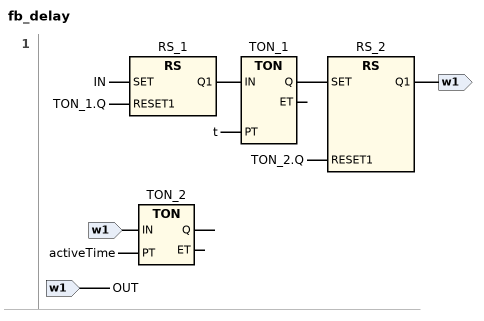
// NETWORK 1
RS_1(SET := IN, RESET1 := TON_1.Q); // RS
TON_1(IN := RS_1.Q1, PT := t); // TON
RS_2(SET := TON_1.Q, RESET1 := TON_2.Q); // RS
TON_2(IN := RS_2.Q1, PT := activeTime); // TON
OUT := RS_2.Q1;

END_FUNCTION_BLOCK

// Device/Application/functions/FB_CLK
// 50 % CLK heigh
FUNCTION_BLOCK FB_CLK
VAR_INPUT
	enable : BOOL := TRUE;
	CLK_Time : TIME := T#1s;
END_VAR
VAR
	RS_0: RS;
	TON_0: TON;
	RS_1: RS;
	TON_1: TON;
END_VAR
VAR_OUTPUT
	CLK :BOOL;
END_VAR

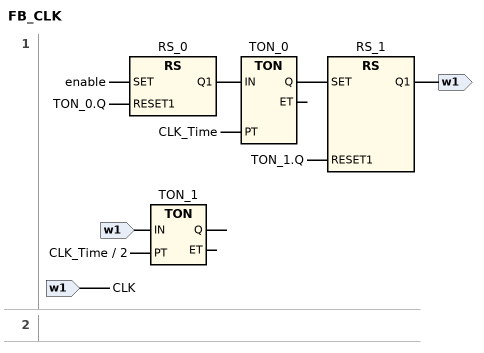
// NETWORK 1
RS_0(SET := enable, RESET1 := TON_0.Q); // RS
TON_0(IN := RS_0.Q1, PT := CLK_Time); // TON
RS_1(SET := TON_0.Q, RESET1 := TON_1.Q); // RS
TON_1(IN := RS_1.Q1, PT := CLK_Time / 2); // TON
CLK := RS_1.Q1;

// NETWORK 2

END_FUNCTION_BLOCK

// Device/Application/functions/Advanced_CTUD
FUNCTION_BLOCK Advanced_CTUD
VAR_INPUT
	CU: BOOL; //key
	CD: BOOL; //key
	activate: BOOL; // exmaple: index = 3 then true.
	frame: USINT; // frame where the button is
	reset : BOOL := 0; // reset to countValue before submit
	//submit : BOOL:= TRUE; // currently not working key or anything else, you can use trigger to make countedValue = newValue
	minValue : INT;
	maxValue: INT;
	countedValue: UINT;
END_VAR
VAR_OUTPUT
	newValue: UINT;
	active : BOOL;
END_VAR
VAR
	FB_smoothCLK_CU: FB_smoothCLK;
	FB_smoothCLK_CD: FB_smoothCLK;
	CTUD_Value: CTUD;
	SR_Changed: SR;
	MIN_1: BOOL;
END_VAR

VAR_IN_OUT

END_VAR
VAR // added by the converter: edge detectors and wires of the graphical bodies
    _rt1, _rt2, _rt3, _rt4, _rt5, _rt6, _rt7 : R_TRIG;
END_VAR

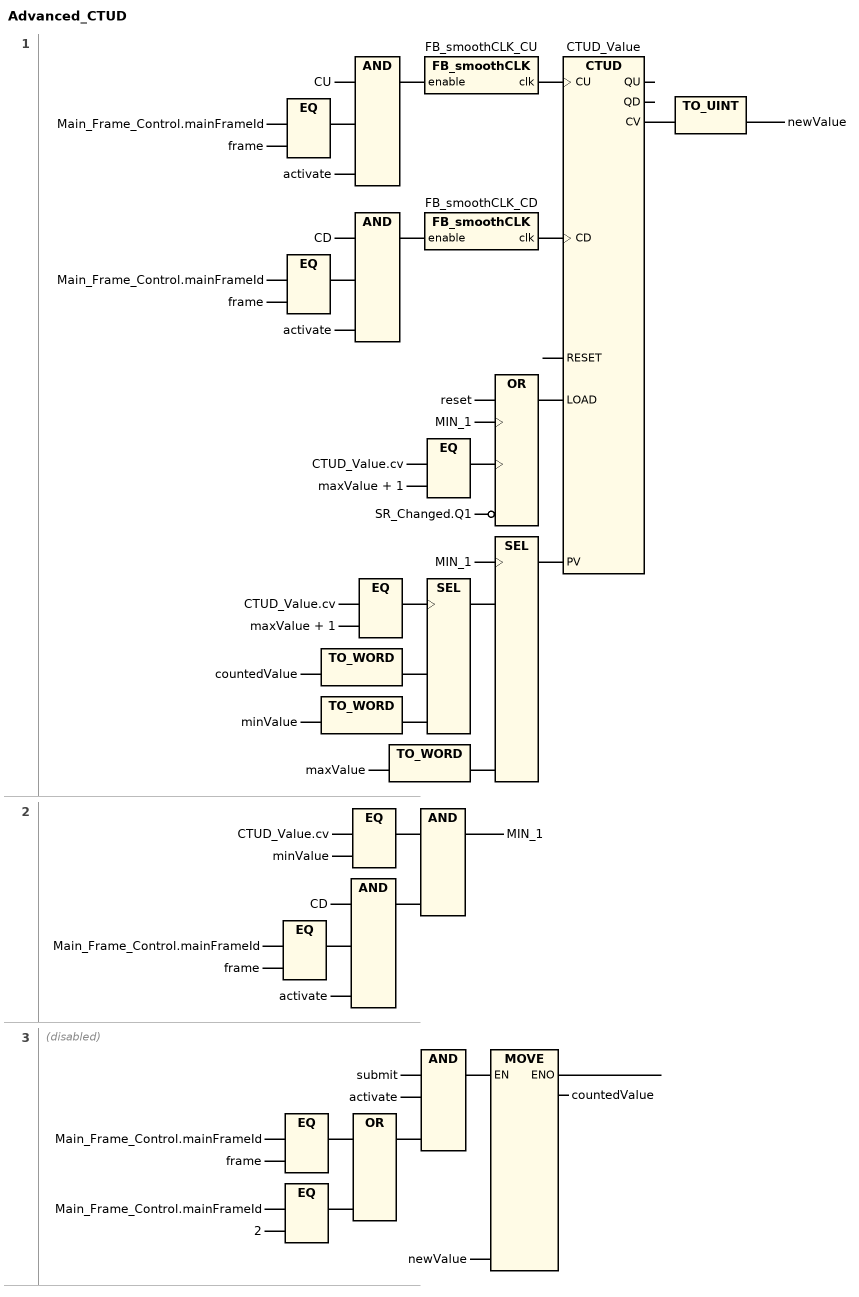
// NETWORK 1
FB_smoothCLK_CU(enable := CU AND Main_Frame_Control.mainFrameId = frame AND activate); // FB_smoothCLK
_rt1(CLK := FB_smoothCLK_CU.clk);
FB_smoothCLK_CD(enable := CD AND Main_Frame_Control.mainFrameId = frame AND activate); // FB_smoothCLK
_rt2(CLK := FB_smoothCLK_CD.clk);
_rt3(CLK := MIN_1);
_rt4(CLK := CTUD_Value.cv = (maxValue + 1));
_rt5(CLK := MIN_1);
_rt6(CLK := CTUD_Value.cv = (maxValue + 1));
CTUD_Value(
    CU := _rt1.Q,
    CD := _rt2.Q,
    LOAD := reset OR _rt3.Q OR _rt4.Q OR NOT SR_Changed.Q1,
    PV := SEL(_rt5.Q, SEL(_rt6.Q, TO_WORD(countedValue), TO_WORD(minValue)), TO_WORD(maxValue))); // CTUD
newValue := TO_UINT(CTUD_Value.CV);

// NETWORK 2
MIN_1 := CTUD_Value.cv = minValue AND (CD AND Main_Frame_Control.mainFrameId = frame AND activate);

// NETWORK 3 (disabled)
// IF submit AND activate AND (Main_Frame_Control.mainFrameId = frame OR Main_Frame_Control.mainFrameId = 2) THEN
//     countedValue := newValue;
// END_IF

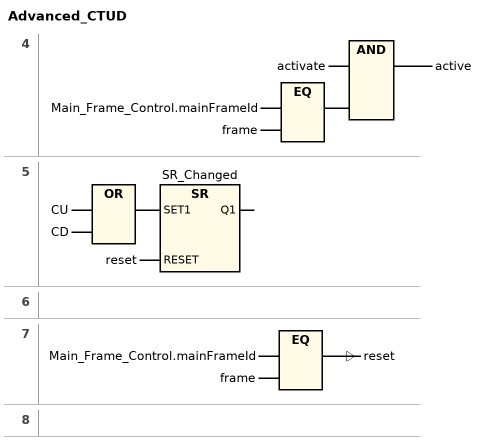
// NETWORK 4
active := activate AND Main_Frame_Control.mainFrameId = frame;

// NETWORK 5
SR_Changed(SET1 := CU OR CD, RESET := reset); // SR

// NETWORK 6

// NETWORK 7
_rt7(CLK := Main_Frame_Control.mainFrameId = frame);
reset := _rt7.Q;

// NETWORK 8

END_FUNCTION_BLOCK

// Device/Application/functions/FB_smoothCLK
FUNCTION_BLOCK FB_smoothCLK
VAR_INPUT
	enable : BOOL := TRUE; // use the same variable wich you used to In- or decrement the value
	CLK_TimeMin : TIME := T#50MS;
	//v : TIME := T#100MS; // sekund^-1
END_VAR
VAR_OUTPUT
	clk: BOOL;
END_VAR
VAR
	FB_CLK_0: FB_CLK;
	CLK_Time: TIME := T#1000MS;
	CLK_Time_End: TIME;
	FB_CLK_1: FB_CLK;
END_VAR
VAR // added by the converter: edge detectors and wires of the graphical bodies
    _w1 : INT;
    _ft1 : F_TRIG;
END_VAR

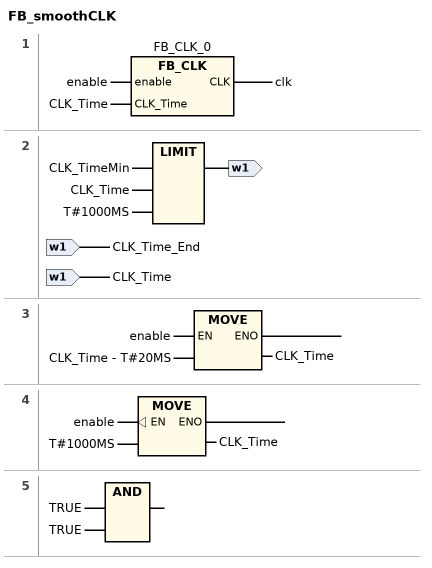
// NETWORK 1
FB_CLK_0(enable := enable, CLK_Time := CLK_Time); // FB_CLK
clk := FB_CLK_0.CLK;

// NETWORK 2
_w1 := LIMIT(CLK_TimeMin, CLK_Time, T#1000MS);
CLK_Time_End := _w1;
CLK_Time := _w1;

// NETWORK 3
IF enable THEN CLK_Time := CLK_Time - T#20MS; END_IF

// NETWORK 4
_ft1(CLK := enable);
IF _ft1.Q THEN CLK_Time := T#1000MS; END_IF

// NETWORK 5
(* TRUE AND TRUE; result not used *)

END_FUNCTION_BLOCK

// Device/Application/FBs/Paramater/parameterUpdate
FUNCTION_BLOCK parameterUpdate
VAR_INPUT
	EN: BOOL;
	selectedParameterIndex: INT;
END_VAR
VAR_OUTPUT


	iDistanceBetweenRowsInMeter: REAL:= 1.5;
	iDistanceBeforInMeter: REAL:= 1.5;
	iDistanceAfterInMeter: REAL:= 1.5;
	iCountRows: USINT:=15 ;
	strRowsDirection: STRING;
	bRowsDirection: BOOL;
	
END_VAR
VAR
	CTU_LeftRight: CTU;
	FB_ChangeDistance_CountRows: FB_UpdatingDistanceParameter;
	FB_ChangeDistance_AfterInMeter: FB_UpdatingDistanceParameter;
	FB_ChangeDistance_BeforInMeter: FB_UpdatingDistanceParameter;
	FB_ChangeDistance_BetweenInMeter: FB_UpdatingDistanceParameter;
	rCountRows: REAL;
	TOGGLE_0:TOGGLE;
	TON_CLK: TON;
	RS_CLK: RS;

	// Row Parameter

	CLK_PULSE_0: CLK_PULSE;
	RS_CLK2: RS;
	TON_CLK2: TON;
END_VAR

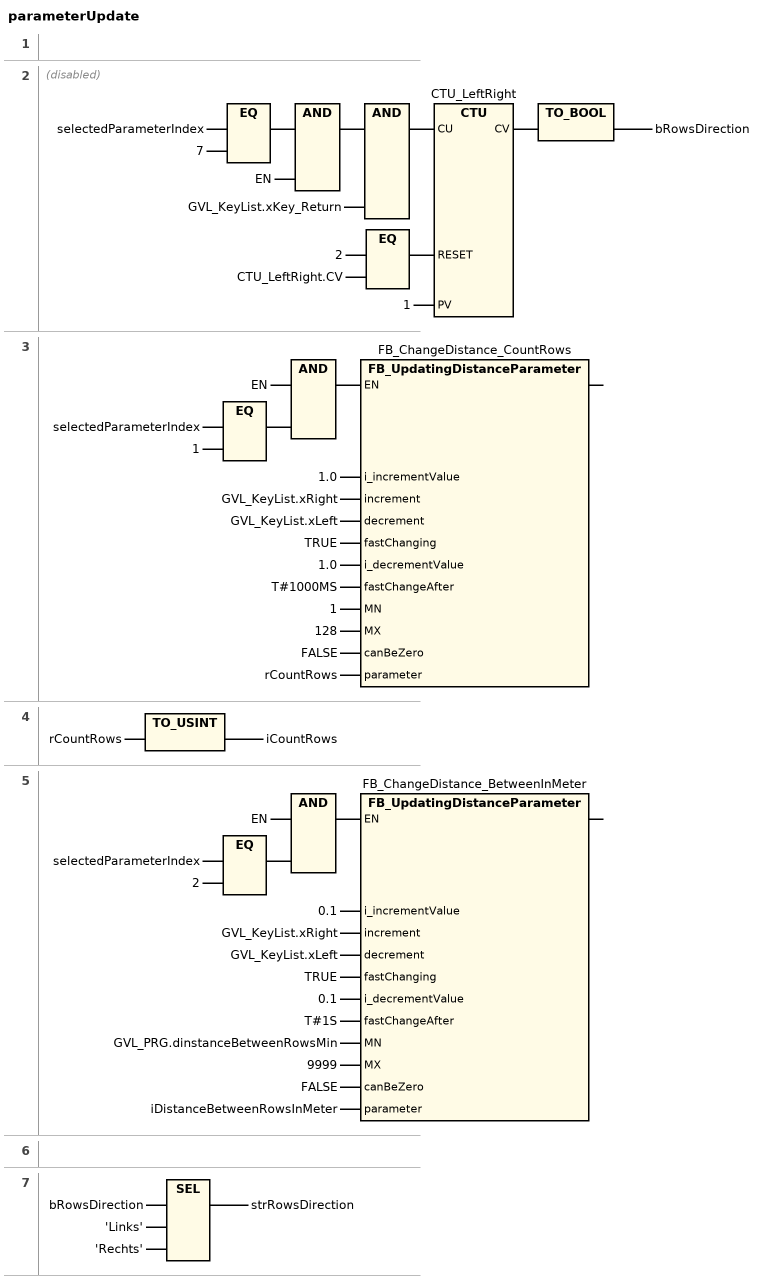
// NETWORK 1

// NETWORK 2 (disabled)
// CTU_LeftRight(
//     CU := (selectedParameterIndex = 7 AND EN) AND GVL_KeyList.xKey_Return,
//     RESET := 2 = CTU_LeftRight.CV,
//     PV := 1); // CTU
// bRowsDirection := TO_BOOL(CTU_LeftRight.CV);

// NETWORK 3
FB_ChangeDistance_CountRows(
    EN := EN AND selectedParameterIndex = 1,
    i_incrementValue := 1.0,
    increment := GVL_KeyList.xRight,
    decrement := GVL_KeyList.xLeft,
    fastChanging := TRUE,
    i_decrementValue := 1.0,
    fastChangeAfter := T#1000MS,
    MN := 1,
    MX := 128,
    canBeZero := FALSE,
    parameter := rCountRows); // FB_UpdatingDistanceParameter

// NETWORK 4
iCountRows := TO_USINT(rCountRows);

// NETWORK 5
FB_ChangeDistance_BetweenInMeter(
    EN := EN AND selectedParameterIndex = 2,
    i_incrementValue := 0.1,
    increment := GVL_KeyList.xRight,
    decrement := GVL_KeyList.xLeft,
    fastChanging := TRUE,
    i_decrementValue := 0.1,
    fastChangeAfter := T#1S,
    MN := GVL_PRG.dinstanceBetweenRowsMin,
    MX := 9999,
    canBeZero := FALSE,
    parameter := iDistanceBetweenRowsInMeter); // FB_UpdatingDistanceParameter

// NETWORK 6

// NETWORK 7
strRowsDirection := SEL(bRowsDirection, 'Links', 'Rechts');

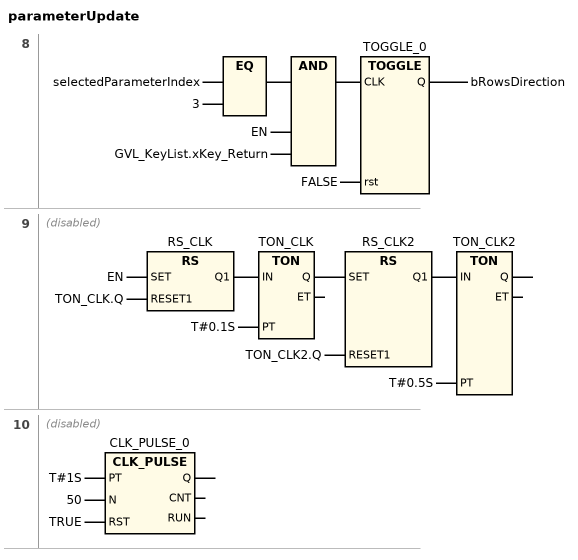
// NETWORK 8
TOGGLE_0(CLK := selectedParameterIndex = 3 AND EN AND GVL_KeyList.xKey_Return, rst := FALSE); // TOGGLE
bRowsDirection := TOGGLE_0.Q;

// NETWORK 9 (disabled)
// RS_CLK(SET := EN, RESET1 := TON_CLK.Q); // RS
// TON_CLK(IN := RS_CLK.Q1, PT := T#0.1S); // TON
// RS_CLK2(SET := TON_CLK.Q, RESET1 := TON_CLK2.Q); // RS
// TON_CLK2(IN := RS_CLK2.Q1, PT := T#0.5S); // TON

// NETWORK 10 (disabled)
// CLK_PULSE_0(PT := T#1S, N := 50, RST := TRUE); // CLK_PULSE

END_FUNCTION_BLOCK

// Device/Application/FBs/Paramater/FB_UpdatingDistanceParameter
FUNCTION_BLOCK FB_UpdatingDistanceParameter
VAR_INPUT
	EN: BOOL;
	i_incrementValue: REAL := 0.1;
	increment: BOOL := FALSE;
	decrement: BOOL := FALSE;
	fastChanging: BOOL := TRUE;
	i_decrementValue: REAL := 0.1;
	fastChangeAfter: TIME:= T#1S;
	MN: REAL := 0;
	MX: REAL:= 9999;
	canBeZero: BOOL:= TRUE;
	
END_VAR
VAR_OUTPUT
END_VAR
VAR
	RS_CLK: RS;
	TON_CLK: TON;
	canBeZeroIfMnGreaterO: BOOL;
	TON_FastEditingDown: TON;
	TON_FastEditingUp: TON;
	canBeZeroIfMXLessThan0: BOOL;
	incrementValue: REAL;
	decrementValue: REAL;
END_VAR
VAR_IN_OUT
		parameter: REAL;
END_VAR
VAR // added by the converter: edge detectors and wires of the graphical bodies
    _w1, _w2, _w3, _w4 : BOOL;
    _rt1, _rt2, _rt3, _rt4 : R_TRIG;
END_VAR

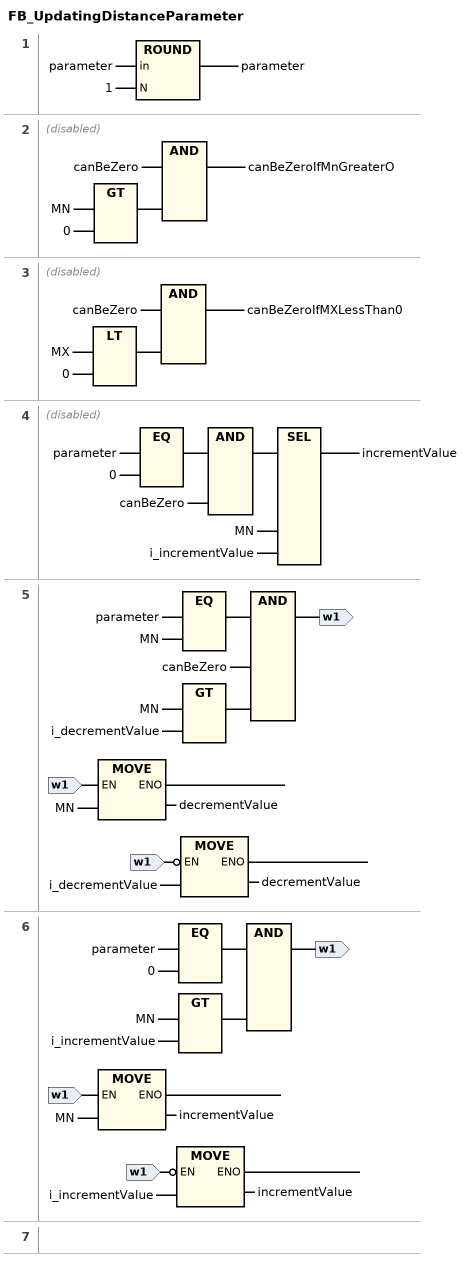
// NETWORK 1
parameter := ROUND(in := parameter, N := 1);

// NETWORK 2 (disabled)
// canBeZeroIfMnGreaterO := canBeZero AND MN > 0;

// NETWORK 3 (disabled)
// canBeZeroIfMXLessThan0 := canBeZero AND MX < 0;

// NETWORK 4 (disabled)
// incrementValue := SEL(parameter = 0 AND canBeZero, MN, i_incrementValue);

// NETWORK 5
_w1 := parameter = MN AND canBeZero AND MN > i_decrementValue;
IF _w1 THEN decrementValue := MN; END_IF
IF NOT _w1 THEN decrementValue := i_decrementValue; END_IF

// NETWORK 6
_w2 := parameter = 0 AND MN > i_incrementValue;
IF _w2 THEN incrementValue := MN; END_IF
IF NOT _w2 THEN incrementValue := i_incrementValue; END_IF

// NETWORK 7

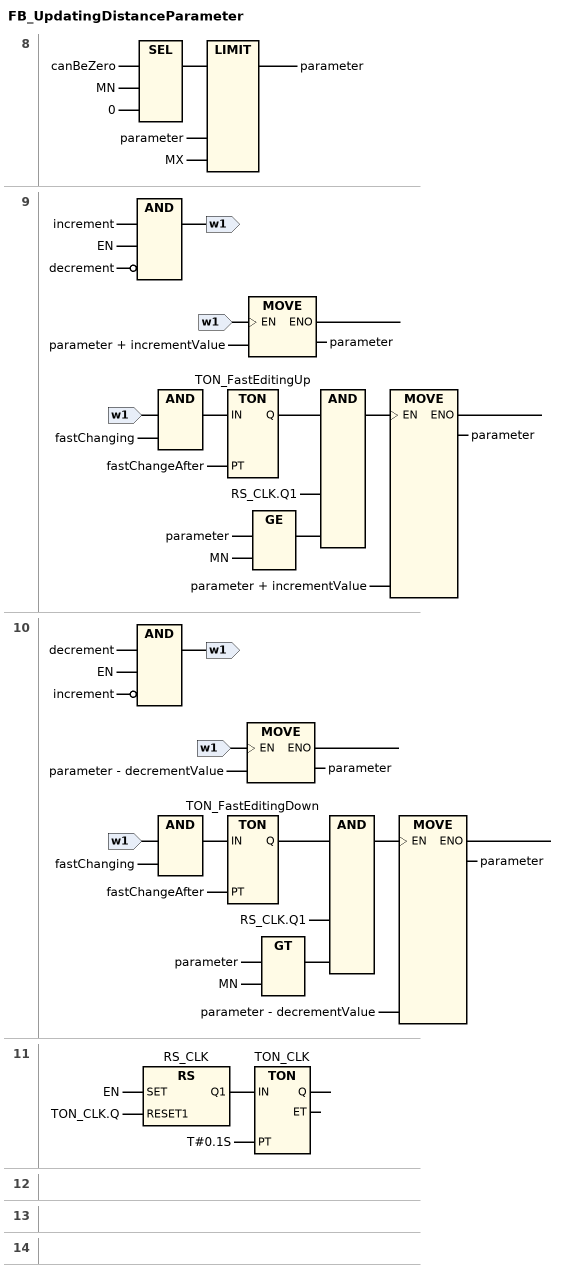
// NETWORK 8
parameter := LIMIT(SEL(canBeZero, MN, 0), parameter, MX);

// NETWORK 9
_w3 := increment AND EN AND NOT decrement;
_rt1(CLK := _w3);
IF _rt1.Q THEN parameter := parameter + incrementValue; END_IF
TON_FastEditingUp(IN := _w3 AND fastChanging, PT := fastChangeAfter); // TON
_rt2(CLK := TON_FastEditingUp.Q AND RS_CLK.Q1 AND parameter >= MN);
IF _rt2.Q THEN parameter := parameter + incrementValue; END_IF

// NETWORK 10
_w4 := decrement AND EN AND NOT increment;
_rt3(CLK := _w4);
IF _rt3.Q THEN parameter := parameter - decrementValue; END_IF
TON_FastEditingDown(IN := _w4 AND fastChanging, PT := fastChangeAfter); // TON
_rt4(CLK := TON_FastEditingDown.Q AND RS_CLK.Q1 AND parameter > MN);
IF _rt4.Q THEN parameter := parameter - decrementValue; END_IF

// NETWORK 11
RS_CLK(SET := EN, RESET1 := TON_CLK.Q); // RS
TON_CLK(IN := RS_CLK.Q1, PT := T#0.1S); // TON

// NETWORK 12

// NETWORK 13

// NETWORK 14

END_FUNCTION_BLOCK

// Device/Application/FBs/Controll/RoboterControl
FUNCTION_BLOCK RoboterControl
VAR_INPUT
	
	iCountRows:USINT;
	iDistanceAfterInMeter: REAL;
	iDistanceBeforInMeter: REAL;
	iDistanceBetweenRowsInMeter: REAL;
	bRowsDirection: BOOL;
END_VAR
VAR_OUTPUT
END_VAR
VAR
	AutomaticModeControl_0: AutomaticModeControl;
	PrepareAutomaticModeParameterForCAN_0: PrepareParameterForCAN;
END_VAR
VAR // added by the converter: edge detectors and wires of the graphical bodies
    _rt1, _rt2 : R_TRIG;
END_VAR

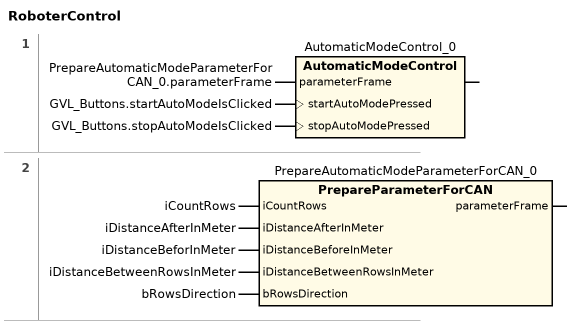
// NETWORK 1
_rt1(CLK := GVL_Buttons.startAutoModeIsClicked);
_rt2(CLK := GVL_Buttons.stopAutoModeIsClicked);
AutomaticModeControl_0(
    parameterFrame := PrepareAutomaticModeParameterForCAN_0.parameterFrame,
    startAutoModePressed := _rt1.Q,
    stopAutoModePressed := _rt2.Q); // AutomaticModeControl

// NETWORK 2
PrepareAutomaticModeParameterForCAN_0(
    iCountRows := iCountRows,
    iDistanceAfterInMeter := iDistanceAfterInMeter,
    iDistanceBeforeInMeter := iDistanceBeforInMeter,
    iDistanceBetweenRowsInMeter := iDistanceBetweenRowsInMeter,
    bRowsDirection := bRowsDirection); // PrepareParameterForCAN

END_FUNCTION_BLOCK

// Device/Application/FBs/Controll/AutomaticModeControl
FUNCTION_BLOCK AutomaticModeControl
VAR_INPUT
	parameterFrame: ARRAY[0..7] OF USINT;
	startAutoModePressed: BOOL;
	stopAutoModePressed: BOOL;
END_VAR
VAR_OUTPUT
END_VAR
VAR
	CAN_Tx_StartAutomode: ifmRCAN.CAN_Tx;
	CAN_Tx_StopAutoMode: ifmRCAN.CAN_Tx;
	CAN_Tx_PauseAutoMode: ifmRCAN.CAN_Tx;
	CAN_Tx_ResumeAutoMode: ifmRCAN.CAN_Tx;
	//AM_Paused: BOOL;
	CAN_Tx_ACK_Stop: ifmRCAN.CAN_Tx;
	SR_0: SR;
	SR_1: SR;
	rs_33: rs;
	CAN_Rx_jetson : ifmRCAN.CAN_Rx;
	SR_start_TX_State_Done: sr;
	fb_delay_1: FB_DELAY;
	FB_CLK_0: FB_CLK;
	test: BOOL;
	test1: BOOL;
	test2: BOOL;
	test4: BOOL;
	SR_waitingStartTime: sr;
	startNow: BOOL;
	test6: BOOL;
END_VAR
VAR // added by the converter: edge detectors and wires of the graphical bodies
    _rt1, _rt2, _rt3, _rt4, _rt5, _rt6, _rt7, _rt8, _rt9, _rt10, _rt11, _rt12, _rt13, _rt14 : R_TRIG;
    _ft1, _ft2, _ft3, _ft4, _ft5, _ft6, _ft7 : F_TRIG;
    _w1, _w2, _w3 : BOOL;
END_VAR

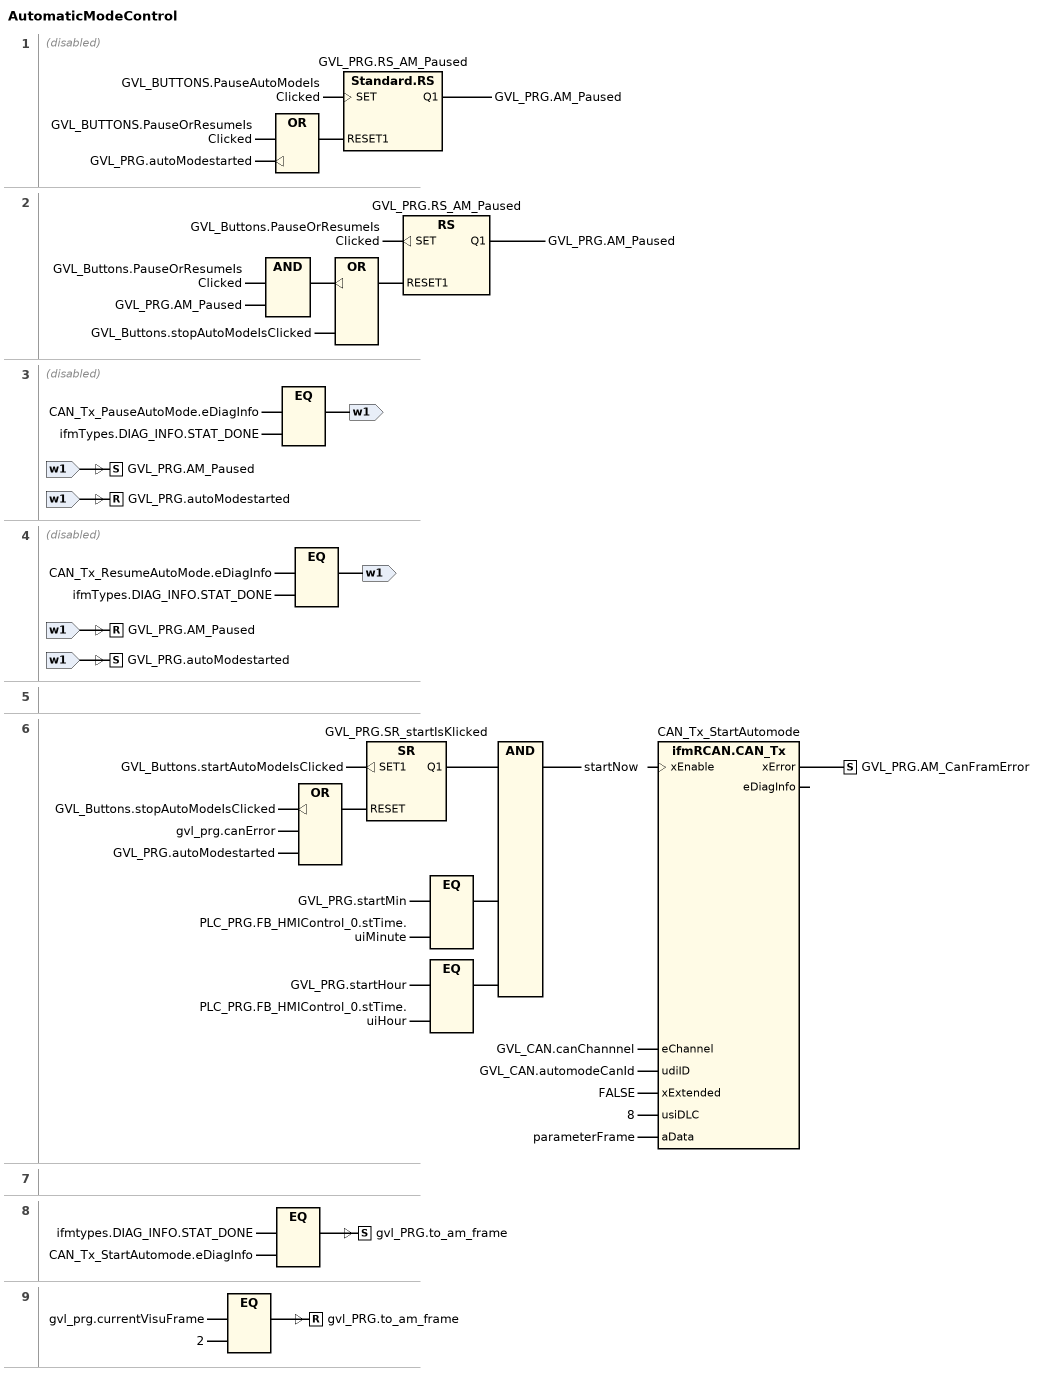
// NETWORK 1 (disabled)
// _rt1(CLK := GVL_BUTTONS.PauseAutoModeIsClicked);
// _ft1(CLK := GVL_PRG.autoModestarted);
// GVL_PRG.RS_AM_Paused(SET := _rt1.Q, RESET1 := GVL_BUTTONS.PauseOrResumeIsClicked OR _ft1.Q); // Standard.RS
// GVL_PRG.AM_Paused := GVL_PRG.RS_AM_Paused.Q1;

// NETWORK 2
_ft2(CLK := GVL_Buttons.PauseOrResumeIsClicked);
_ft3(CLK := GVL_Buttons.PauseOrResumeIsClicked AND GVL_PRG.AM_Paused);
GVL_PRG.RS_AM_Paused(SET := _ft2.Q, RESET1 := _ft3.Q OR GVL_Buttons.stopAutoModeIsClicked); // RS
GVL_PRG.AM_Paused := GVL_PRG.RS_AM_Paused.Q1;

// NETWORK 3 (disabled)
// _w1 := CAN_Tx_PauseAutoMode.eDiagInfo = ifmTypes.DIAG_INFO.STAT_DONE;
// _rt2(CLK := _w1);
// GVL_PRG.AM_Paused S= _rt2.Q;
// _rt3(CLK := _w1);
// GVL_PRG.autoModestarted R= _rt3.Q;

// NETWORK 4 (disabled)
// _w2 := CAN_Tx_ResumeAutoMode.eDiagInfo = ifmTypes.DIAG_INFO.STAT_DONE;
// _rt4(CLK := _w2);
// GVL_PRG.AM_Paused R= _rt4.Q;
// _rt5(CLK := _w2);
// GVL_PRG.autoModestarted S= _rt5.Q;

// NETWORK 5

// NETWORK 6
_ft4(CLK := GVL_Buttons.startAutoModeIsClicked);
_ft5(CLK := GVL_Buttons.stopAutoModeIsClicked);
GVL_PRG.SR_startIsKlicked(SET1 := _ft4.Q, RESET := _ft5.Q OR gvl_prg.canError OR GVL_PRG.autoModestarted); // SR
_w3 := GVL_PRG.SR_startIsKlicked.Q1 AND GVL_PRG.startMin = PLC_PRG.FB_HMIControl_0.stTime.uiMinute AND GVL_PRG.startHour = PLC_PRG.FB_HMIControl_0.stTime.uiHour;
startNow := _w3;
_rt6(CLK := _w3);
CAN_Tx_StartAutomode(
    xEnable := _rt6.Q,
    eChannel := GVL_CAN.canChannnel,
    udiID := GVL_CAN.automodeCanId,
    xExtended := FALSE,
    usiDLC := 8,
    aData := parameterFrame); // ifmRCAN.CAN_Tx
GVL_PRG.AM_CanFramError S= CAN_Tx_StartAutomode.xError;

// NETWORK 7

// NETWORK 8
_rt7(CLK := ifmtypes.DIAG_INFO.STAT_DONE = CAN_Tx_StartAutomode.eDiagInfo);
gvl_PRG.to_am_frame S= _rt7.Q;

// NETWORK 9
_rt8(CLK := gvl_prg.currentVisuFrame = 2);
gvl_PRG.to_am_frame R= _rt8.Q;

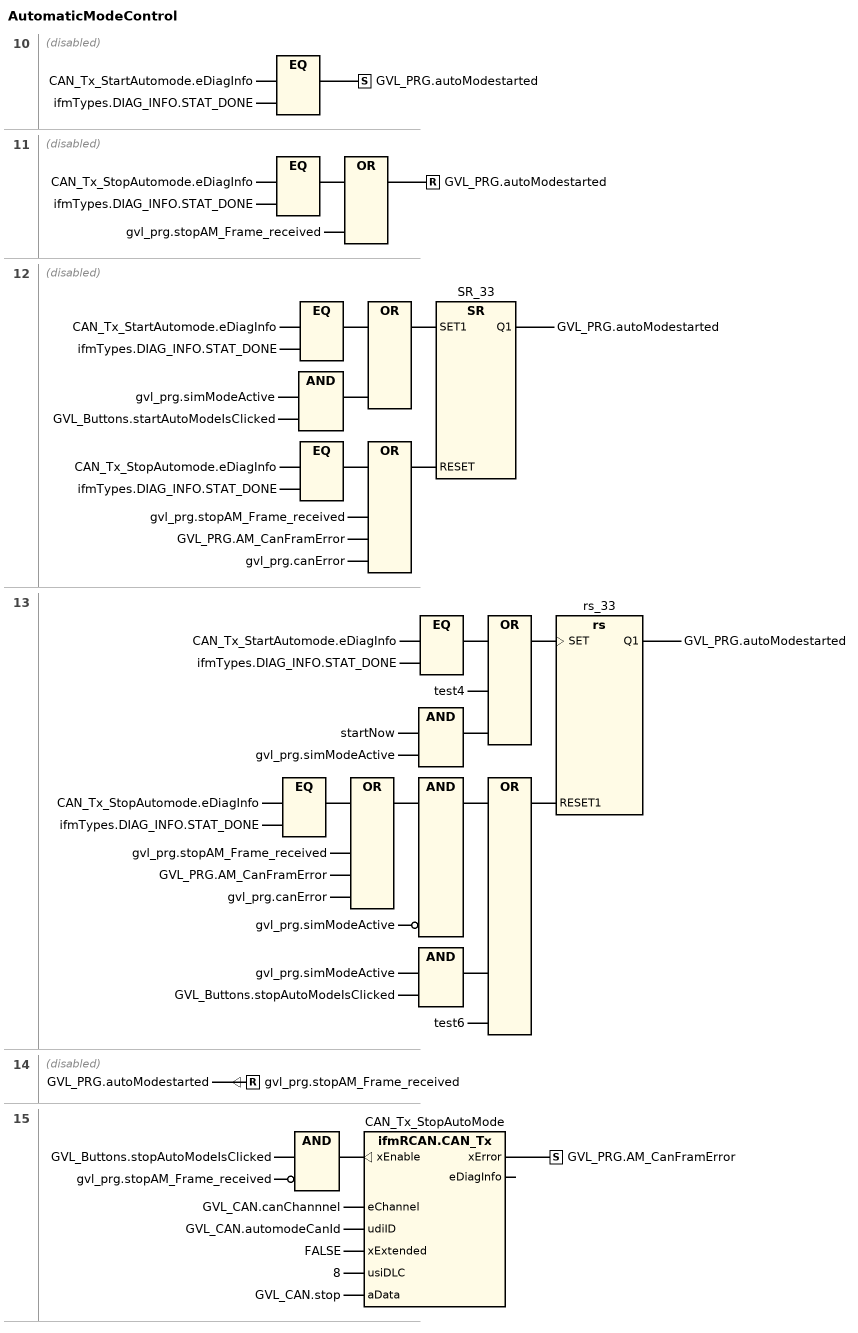
// NETWORK 10 (disabled)
// GVL_PRG.autoModestarted S= CAN_Tx_StartAutomode.eDiagInfo = ifmTypes.DIAG_INFO.STAT_DONE;

// NETWORK 11 (disabled)
// GVL_PRG.autoModestarted R= CAN_Tx_StopAutomode.eDiagInfo = ifmTypes.DIAG_INFO.STAT_DONE OR gvl_prg.stopAM_Frame_received;

// NETWORK 12 (disabled)
// SR_33(SET1 := CAN_Tx_StartAutomode.eDiagInfo = ifmTypes.DIAG_INFO.STAT_DONE OR gvl_prg.simModeActive AND GVL_Buttons.startAutoModeIsClicked, RESET := CAN_Tx_StopAutomode.eDiagInfo = ifmTypes.DIAG_INFO.STAT_DONE OR gvl_prg.stopAM_Frame_received OR GVL_PRG.AM_CanFramError OR gvl_prg.canError); // SR
// GVL_PRG.autoModestarted := SR_33.Q1;

// NETWORK 13
_rt9(CLK := CAN_Tx_StartAutomode.eDiagInfo = ifmTypes.DIAG_INFO.STAT_DONE OR test4 OR startNow AND gvl_prg.simModeActive);
rs_33(SET := _rt9.Q, RESET1 := (CAN_Tx_StopAutomode.eDiagInfo = ifmTypes.DIAG_INFO.STAT_DONE OR gvl_prg.stopAM_Frame_received OR GVL_PRG.AM_CanFramError OR gvl_prg.canError) AND NOT gvl_prg.simModeActive OR gvl_prg.simModeActive AND GVL_Buttons.stopAutoModeIsClicked OR test6); // rs
GVL_PRG.autoModestarted := rs_33.Q1;

// NETWORK 14 (disabled)
// _ft6(CLK := GVL_PRG.autoModestarted);
// gvl_prg.stopAM_Frame_received R= _ft6.Q;

// NETWORK 15
_ft7(CLK := GVL_Buttons.stopAutoModeIsClicked AND NOT gvl_prg.stopAM_Frame_received);
CAN_Tx_StopAutoMode(
    xEnable := _ft7.Q,
    eChannel := GVL_CAN.canChannnel,
    udiID := GVL_CAN.automodeCanId,
    xExtended := FALSE,
    usiDLC := 8,
    aData := GVL_CAN.stop); // ifmRCAN.CAN_Tx
GVL_PRG.AM_CanFramError S= CAN_Tx_StopAutoMode.xError;

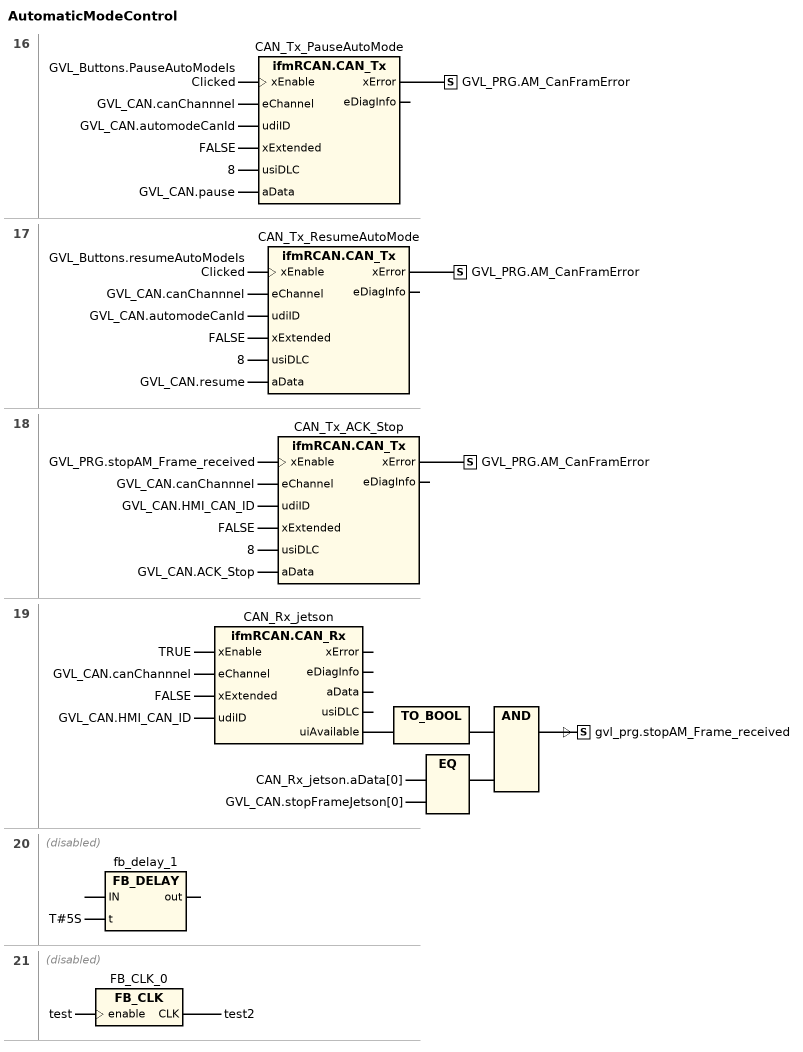
// NETWORK 16
_rt10(CLK := GVL_Buttons.PauseAutoModeIsClicked);
CAN_Tx_PauseAutoMode(
    xEnable := _rt10.Q,
    eChannel := GVL_CAN.canChannnel,
    udiID := GVL_CAN.automodeCanId,
    xExtended := FALSE,
    usiDLC := 8,
    aData := GVL_CAN.pause); // ifmRCAN.CAN_Tx
GVL_PRG.AM_CanFramError S= CAN_Tx_PauseAutoMode.xError;

// NETWORK 17
_rt11(CLK := GVL_Buttons.resumeAutoModeIsClicked);
CAN_Tx_ResumeAutoMode(
    xEnable := _rt11.Q,
    eChannel := GVL_CAN.canChannnel,
    udiID := GVL_CAN.automodeCanId,
    xExtended := FALSE,
    usiDLC := 8,
    aData := GVL_CAN.resume); // ifmRCAN.CAN_Tx
GVL_PRG.AM_CanFramError S= CAN_Tx_ResumeAutoMode.xError;

// NETWORK 18
_rt12(CLK := GVL_PRG.stopAM_Frame_received);
CAN_Tx_ACK_Stop(
    xEnable := _rt12.Q,
    eChannel := GVL_CAN.canChannnel,
    udiID := GVL_CAN.HMI_CAN_ID,
    xExtended := FALSE,
    usiDLC := 8,
    aData := GVL_CAN.ACK_Stop); // ifmRCAN.CAN_Tx
GVL_PRG.AM_CanFramError S= CAN_Tx_ACK_Stop.xError;

// NETWORK 19
CAN_Rx_jetson(
    xEnable := TRUE,
    eChannel := GVL_CAN.canChannnel,
    xExtended := FALSE,
    udiID := GVL_CAN.HMI_CAN_ID); // ifmRCAN.CAN_Rx
_rt13(CLK := TO_BOOL(CAN_Rx_jetson.uiAvailable) AND CAN_Rx_jetson.aData[0] = GVL_CAN.stopFrameJetson[0]);
gvl_prg.stopAM_Frame_received S= _rt13.Q;

// NETWORK 20 (disabled)
// fb_delay_1(t := T#5S); // FB_DELAY

// NETWORK 21 (disabled)
// _rt14(CLK := test);
// FB_CLK_0(enable := _rt14.Q); // FB_CLK
// test2 := FB_CLK_0.CLK;

END_FUNCTION_BLOCK

// Device/Application/FBs/Paramater/PrepareParameterForCAN
FUNCTION_BLOCK PrepareParameterForCAN
VAR_INPUT
	iCountRows:USINT;
	iDistanceAfterInMeter: REAL;
	iDistanceBeforeInMeter: REAL;
	iDistanceBetweenRowsInMeter: REAL;
	bRowsDirection: BOOL;
END_VAR
VAR_OUTPUT
	parameterFrame: ARRAY[0..7] OF USINT:=[0,0,0,0,0,0,0,0];
END_VAR
VAR
	iDistanceAfterInDM: USINT;
	iDistanceBeforeInDM: USINT;
	iDistanceBetweenRowsInDm: USINT;
	iRowsDirection: USINT;
	TO_ARRAY_Parameter: TO_ArrayOfUsint;
	TO_ArrayOfUsint_0: TO_ArrayOfUsint;
END_VAR

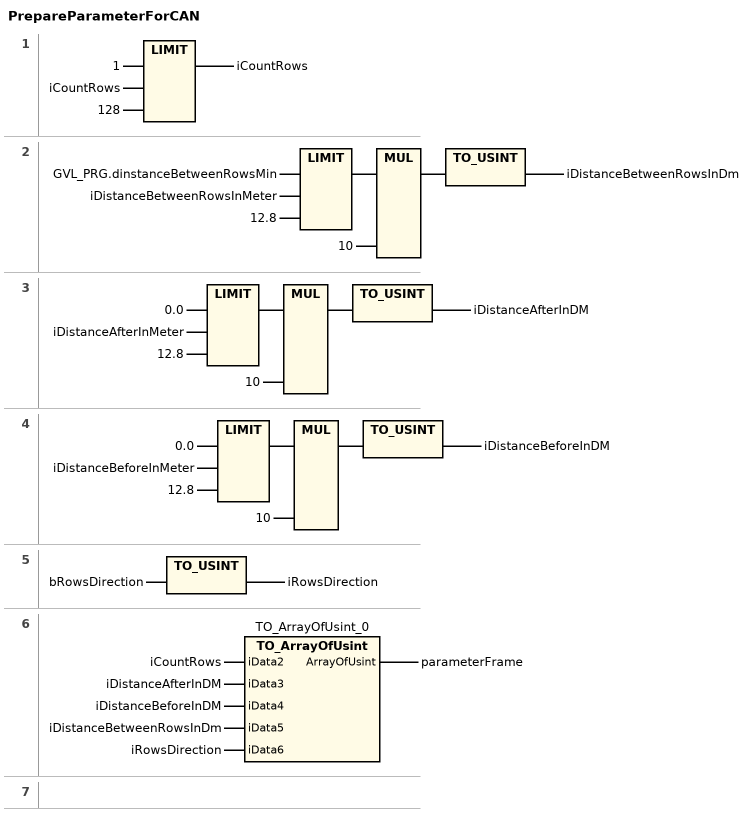
// NETWORK 1
iCountRows := LIMIT(1, iCountRows, 128);

// NETWORK 2
iDistanceBetweenRowsInDm := TO_USINT(LIMIT(GVL_PRG.dinstanceBetweenRowsMin, iDistanceBetweenRowsInMeter, 12.8) * 10);

// NETWORK 3
iDistanceAfterInDM := TO_USINT(LIMIT(0.0, iDistanceAfterInMeter, 12.8) * 10);

// NETWORK 4
iDistanceBeforeInDM := TO_USINT(LIMIT(0.0, iDistanceBeforeInMeter, 12.8) * 10);

// NETWORK 5
iRowsDirection := TO_USINT(bRowsDirection);

// NETWORK 6
TO_ArrayOfUsint_0(
    iData2 := iCountRows,
    iData3 := iDistanceAfterInDM,
    iData4 := iDistanceBeforeInDM,
    iData5 := iDistanceBetweenRowsInDm,
    iData6 := iRowsDirection); // TO_ArrayOfUsint
parameterFrame := TO_ArrayOfUsint_0.ArrayOfUsint;

// NETWORK 7

END_FUNCTION_BLOCK

// Device/Application/FBs/Paramater/TO_ArrayOfUsint
FUNCTION_BLOCK TO_ArrayOfUsint
VAR_INPUT
	iData1 : USINT := 0;
	iData2 : USINT := 0;
	iData3 : USINT := 0;
	iData4 : USINT := 0;
	iData5 : USINT := 0;
	iData6 : USINT := 0;
	iData7 : USINT := 0;
	iData8 : USINT := 0;
END_VAR
VAR_OUTPUT
	ArrayOfUsint: ARRAY [1..8] OF USINT;
END_VAR
VAR
END_VAR

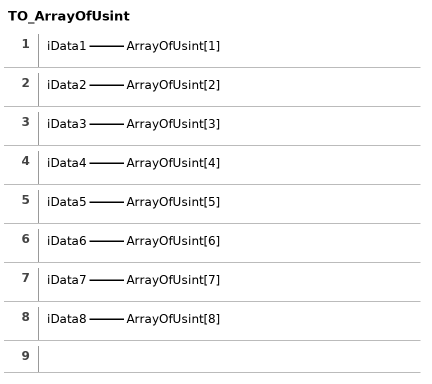
// NETWORK 1
ArrayOfUsint[1] := iData1;

// NETWORK 2
ArrayOfUsint[2] := iData2;

// NETWORK 3
ArrayOfUsint[3] := iData3;

// NETWORK 4
ArrayOfUsint[4] := iData4;

// NETWORK 5
ArrayOfUsint[5] := iData5;

// NETWORK 6
ArrayOfUsint[6] := iData6;

// NETWORK 7
ArrayOfUsint[7] := iData7;

// NETWORK 8
ArrayOfUsint[8] := iData8;

// NETWORK 9

END_FUNCTION_BLOCK

// Device/Application/FBs/Controll/SprayerControl
FUNCTION_BLOCK SprayerControl
VAR_INPUT
	//EN: BOOL;
		selectedParameterIndex: INT;
END_VAR
VAR_OUTPUT
END_VAR
VAR
	CAN_Tx_SprayerStartUp: ifmRCAN.CAN_Tx;
	CAN_Tx_SprayerStopUp: ifmRCAN.CAN_Tx;
	CAN_Tx_SprayerStartDown: ifmRCAN.CAN_Tx;
	CAN_Tx_SprayerStopDown: ifmRCAN.CAN_Tx;

	CAN_Tx_StopSprayer_1: ifmRCAN.CAN_Tx;
	CAN_Tx_StopSprayer_2: ifmRCAN.CAN_Tx;
	CAN_Tx_StopSprayer_3: ifmRCAN.CAN_Tx;
	
	CAN_Tx_PauseSprayer_1: ifmRCAN.CAN_Tx;
	CAN_Tx_PauseSprayer_2: ifmRCAN.CAN_Tx;
	CAN_Tx_PauseSprayer_3: ifmRCAN.CAN_Tx;
	
	CAN_Tx_ResumeSprayer_1: ifmRCAN.CAN_Tx;
	CAN_Tx_ResumeSprayer_2: ifmRCAN.CAN_Tx;
	CAN_Tx_ResumeSprayer_3: ifmRCAN.CAN_Tx;
	CAN_Tx_PumpOn: ifmRCAN.CAN_Tx;
	CAN_Tx_PumpOff: ifmRCAN.CAN_Tx;
	CAN_Tx_spryerLeftOn: ifmRCAN.CAN_Tx;
	CAN_Tx_spryerLeftOff: ifmRCAN.CAN_Tx;
	CAN_Tx_spryerRightOn: ifmRCAN.CAN_Tx;
	CAN_Tx_spryerRightOff: ifmRCAN.CAN_Tx;
END_VAR
VAR // added by the converter: edge detectors and wires of the graphical bodies
    _rt1, _rt2, _rt3, _rt4, _rt5, _rt6, _rt7, _rt8, _rt9, _rt10, _rt11, _rt12, _rt13 : R_TRIG;
    _ft1, _ft2, _ft3, _ft4, _ft5, _ft6 : F_TRIG;
END_VAR

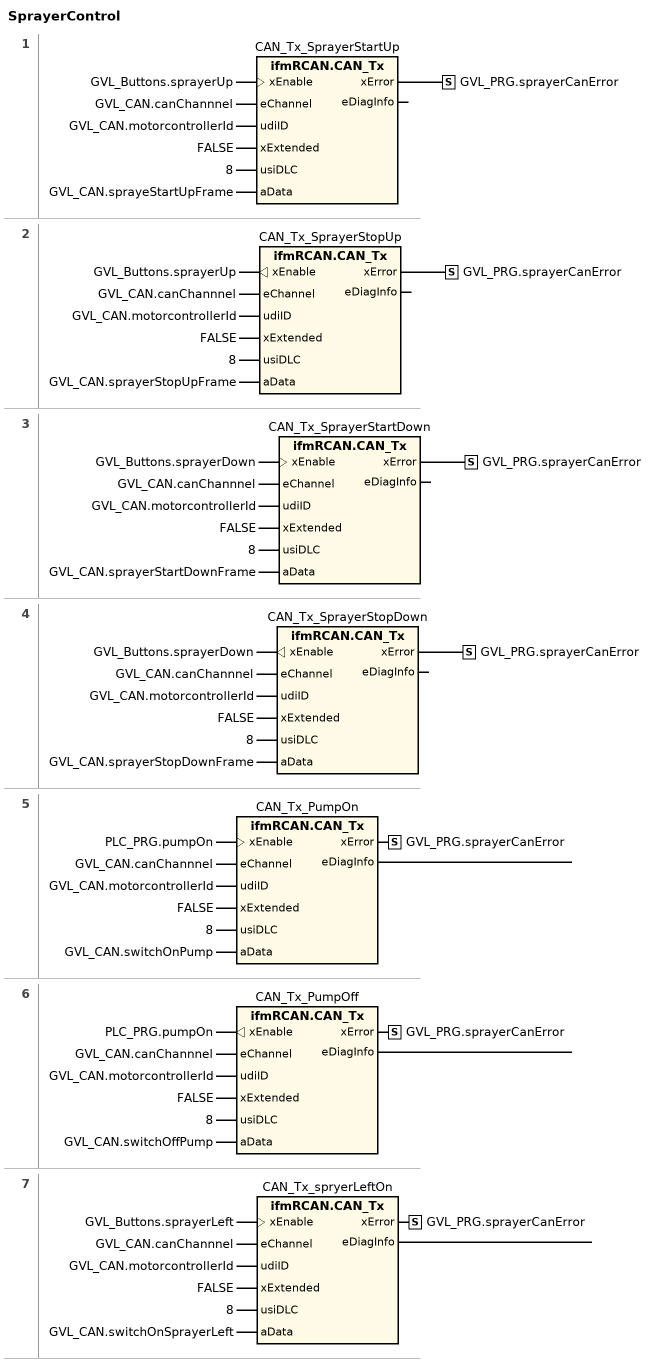
// NETWORK 1
_rt1(CLK := GVL_Buttons.sprayerUp);
CAN_Tx_SprayerStartUp(
    xEnable := _rt1.Q,
    eChannel := GVL_CAN.canChannnel,
    udiID := GVL_CAN.motorcontrollerId,
    xExtended := FALSE,
    usiDLC := 8,
    aData := GVL_CAN.sprayeStartUpFrame); // ifmRCAN.CAN_Tx
GVL_PRG.sprayerCanError S= CAN_Tx_SprayerStartUp.xError;

// NETWORK 2
_ft1(CLK := GVL_Buttons.sprayerUp);
CAN_Tx_SprayerStopUp(
    xEnable := _ft1.Q,
    eChannel := GVL_CAN.canChannnel,
    udiID := GVL_CAN.motorcontrollerId,
    xExtended := FALSE,
    usiDLC := 8,
    aData := GVL_CAN.sprayerStopUpFrame); // ifmRCAN.CAN_Tx
GVL_PRG.sprayerCanError S= CAN_Tx_SprayerStopUp.xError;

// NETWORK 3
_rt2(CLK := GVL_Buttons.sprayerDown);
CAN_Tx_SprayerStartDown(
    xEnable := _rt2.Q,
    eChannel := GVL_CAN.canChannnel,
    udiID := GVL_CAN.motorcontrollerId,
    xExtended := FALSE,
    usiDLC := 8,
    aData := GVL_CAN.sprayerStartDownFrame); // ifmRCAN.CAN_Tx
GVL_PRG.sprayerCanError S= CAN_Tx_SprayerStartDown.xError;

// NETWORK 4
_ft2(CLK := GVL_Buttons.sprayerDown);
CAN_Tx_SprayerStopDown(
    xEnable := _ft2.Q,
    eChannel := GVL_CAN.canChannnel,
    udiID := GVL_CAN.motorcontrollerId,
    xExtended := FALSE,
    usiDLC := 8,
    aData := GVL_CAN.sprayerStopDownFrame); // ifmRCAN.CAN_Tx
GVL_PRG.sprayerCanError S= CAN_Tx_SprayerStopDown.xError;

// NETWORK 5
_rt3(CLK := PLC_PRG.pumpOn);
CAN_Tx_PumpOn(
    xEnable := _rt3.Q,
    eChannel := GVL_CAN.canChannnel,
    udiID := GVL_CAN.motorcontrollerId,
    xExtended := FALSE,
    usiDLC := 8,
    aData := GVL_CAN.switchOnPump); // ifmRCAN.CAN_Tx
GVL_PRG.sprayerCanError S= CAN_Tx_PumpOn.xError;

// NETWORK 6
_ft3(CLK := PLC_PRG.pumpOn);
CAN_Tx_PumpOff(
    xEnable := _ft3.Q,
    eChannel := GVL_CAN.canChannnel,
    udiID := GVL_CAN.motorcontrollerId,
    xExtended := FALSE,
    usiDLC := 8,
    aData := GVL_CAN.switchOffPump); // ifmRCAN.CAN_Tx
GVL_PRG.sprayerCanError S= CAN_Tx_PumpOff.xError;

// NETWORK 7
_rt4(CLK := GVL_Buttons.sprayerLeft);
CAN_Tx_spryerLeftOn(
    xEnable := _rt4.Q,
    eChannel := GVL_CAN.canChannnel,
    udiID := GVL_CAN.motorcontrollerId,
    xExtended := FALSE,
    usiDLC := 8,
    aData := GVL_CAN.switchOnSprayerLeft); // ifmRCAN.CAN_Tx
GVL_PRG.sprayerCanError S= CAN_Tx_spryerLeftOn.xError;

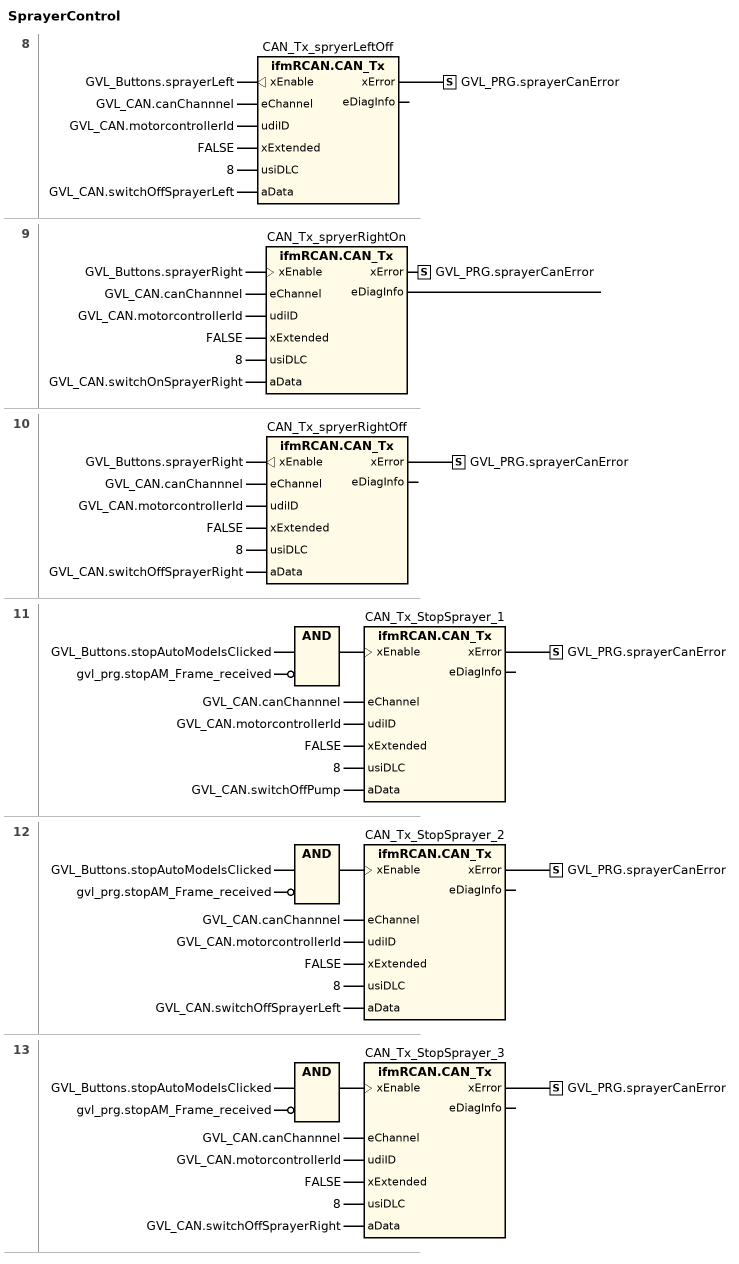
// NETWORK 8
_ft4(CLK := GVL_Buttons.sprayerLeft);
CAN_Tx_spryerLeftOff(
    xEnable := _ft4.Q,
    eChannel := GVL_CAN.canChannnel,
    udiID := GVL_CAN.motorcontrollerId,
    xExtended := FALSE,
    usiDLC := 8,
    aData := GVL_CAN.switchOffSprayerLeft); // ifmRCAN.CAN_Tx
GVL_PRG.sprayerCanError S= CAN_Tx_spryerLeftOff.xError;

// NETWORK 9
_rt5(CLK := GVL_Buttons.sprayerRight);
CAN_Tx_spryerRightOn(
    xEnable := _rt5.Q,
    eChannel := GVL_CAN.canChannnel,
    udiID := GVL_CAN.motorcontrollerId,
    xExtended := FALSE,
    usiDLC := 8,
    aData := GVL_CAN.switchOnSprayerRight); // ifmRCAN.CAN_Tx
GVL_PRG.sprayerCanError S= CAN_Tx_spryerRightOn.xError;

// NETWORK 10
_ft5(CLK := GVL_Buttons.sprayerRight);
CAN_Tx_spryerRightOff(
    xEnable := _ft5.Q,
    eChannel := GVL_CAN.canChannnel,
    udiID := GVL_CAN.motorcontrollerId,
    xExtended := FALSE,
    usiDLC := 8,
    aData := GVL_CAN.switchOffSprayerRight); // ifmRCAN.CAN_Tx
GVL_PRG.sprayerCanError S= CAN_Tx_spryerRightOff.xError;

// NETWORK 11
_rt6(CLK := GVL_Buttons.stopAutoModeIsClicked AND NOT gvl_prg.stopAM_Frame_received);
CAN_Tx_StopSprayer_1(
    xEnable := _rt6.Q,
    eChannel := GVL_CAN.canChannnel,
    udiID := GVL_CAN.motorcontrollerId,
    xExtended := FALSE,
    usiDLC := 8,
    aData := GVL_CAN.switchOffPump); // ifmRCAN.CAN_Tx
GVL_PRG.sprayerCanError S= CAN_Tx_StopSprayer_1.xError;

// NETWORK 12
_rt7(CLK := GVL_Buttons.stopAutoModeIsClicked AND NOT gvl_prg.stopAM_Frame_received);
CAN_Tx_StopSprayer_2(
    xEnable := _rt7.Q,
    eChannel := GVL_CAN.canChannnel,
    udiID := GVL_CAN.motorcontrollerId,
    xExtended := FALSE,
    usiDLC := 8,
    aData := GVL_CAN.switchOffSprayerLeft); // ifmRCAN.CAN_Tx
GVL_PRG.sprayerCanError S= CAN_Tx_StopSprayer_2.xError;

// NETWORK 13
_rt8(CLK := GVL_Buttons.stopAutoModeIsClicked AND NOT gvl_prg.stopAM_Frame_received);
CAN_Tx_StopSprayer_3(
    xEnable := _rt8.Q,
    eChannel := GVL_CAN.canChannnel,
    udiID := GVL_CAN.motorcontrollerId,
    xExtended := FALSE,
    usiDLC := 8,
    aData := GVL_CAN.switchOffSprayerRight); // ifmRCAN.CAN_Tx
GVL_PRG.sprayerCanError S= CAN_Tx_StopSprayer_3.xError;

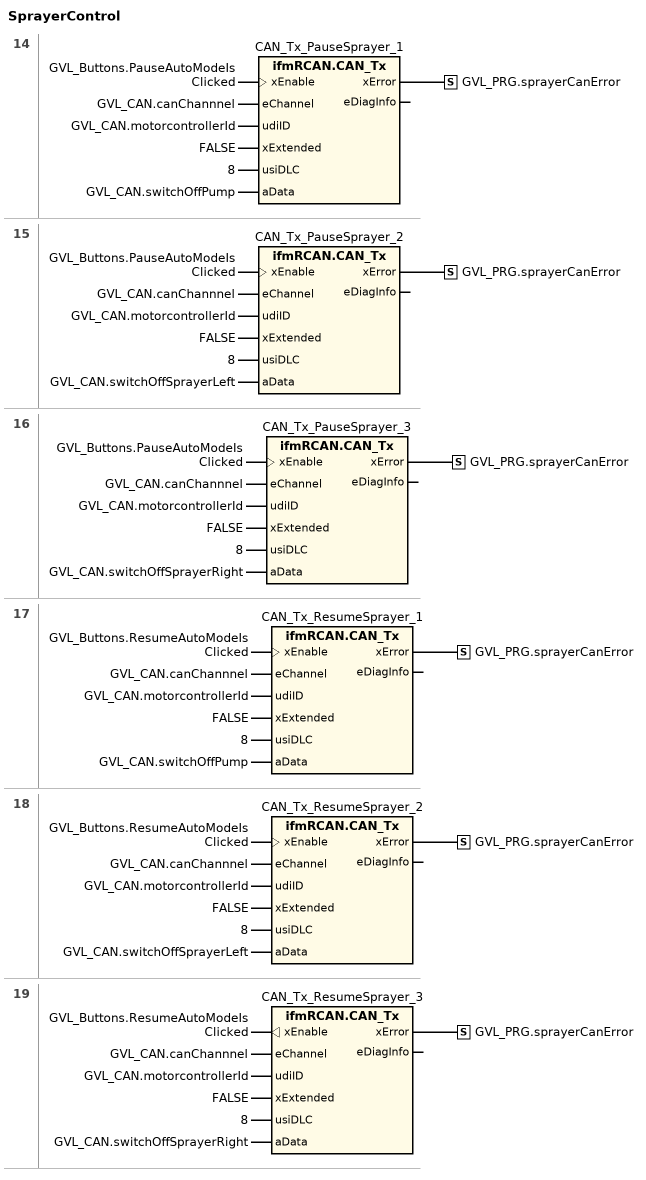
// NETWORK 14
_rt9(CLK := GVL_Buttons.PauseAutoModeIsClicked);
CAN_Tx_PauseSprayer_1(
    xEnable := _rt9.Q,
    eChannel := GVL_CAN.canChannnel,
    udiID := GVL_CAN.motorcontrollerId,
    xExtended := FALSE,
    usiDLC := 8,
    aData := GVL_CAN.switchOffPump); // ifmRCAN.CAN_Tx
GVL_PRG.sprayerCanError S= CAN_Tx_PauseSprayer_1.xError;

// NETWORK 15
_rt10(CLK := GVL_Buttons.PauseAutoModeIsClicked);
CAN_Tx_PauseSprayer_2(
    xEnable := _rt10.Q,
    eChannel := GVL_CAN.canChannnel,
    udiID := GVL_CAN.motorcontrollerId,
    xExtended := FALSE,
    usiDLC := 8,
    aData := GVL_CAN.switchOffSprayerLeft); // ifmRCAN.CAN_Tx
GVL_PRG.sprayerCanError S= CAN_Tx_PauseSprayer_2.xError;

// NETWORK 16
_rt11(CLK := GVL_Buttons.PauseAutoModeIsClicked);
CAN_Tx_PauseSprayer_3(
    xEnable := _rt11.Q,
    eChannel := GVL_CAN.canChannnel,
    udiID := GVL_CAN.motorcontrollerId,
    xExtended := FALSE,
    usiDLC := 8,
    aData := GVL_CAN.switchOffSprayerRight); // ifmRCAN.CAN_Tx
GVL_PRG.sprayerCanError S= CAN_Tx_PauseSprayer_3.xError;

// NETWORK 17
_rt12(CLK := GVL_Buttons.ResumeAutoModeIsClicked);
CAN_Tx_ResumeSprayer_1(
    xEnable := _rt12.Q,
    eChannel := GVL_CAN.canChannnel,
    udiID := GVL_CAN.motorcontrollerId,
    xExtended := FALSE,
    usiDLC := 8,
    aData := GVL_CAN.switchOffPump); // ifmRCAN.CAN_Tx
GVL_PRG.sprayerCanError S= CAN_Tx_ResumeSprayer_1.xError;

// NETWORK 18
_rt13(CLK := GVL_Buttons.ResumeAutoModeIsClicked);
CAN_Tx_ResumeSprayer_2(
    xEnable := _rt13.Q,
    eChannel := GVL_CAN.canChannnel,
    udiID := GVL_CAN.motorcontrollerId,
    xExtended := FALSE,
    usiDLC := 8,
    aData := GVL_CAN.switchOffSprayerLeft); // ifmRCAN.CAN_Tx
GVL_PRG.sprayerCanError S= CAN_Tx_ResumeSprayer_2.xError;

// NETWORK 19
_ft6(CLK := GVL_Buttons.ResumeAutoModeIsClicked);
CAN_Tx_ResumeSprayer_3(
    xEnable := _ft6.Q,
    eChannel := GVL_CAN.canChannnel,
    udiID := GVL_CAN.motorcontrollerId,
    xExtended := FALSE,
    usiDLC := 8,
    aData := GVL_CAN.switchOffSprayerRight); // ifmRCAN.CAN_Tx
GVL_PRG.sprayerCanError S= CAN_Tx_ResumeSprayer_3.xError;

END_FUNCTION_BLOCK

// Device/Application/FBs/Roboter_States/FB_CAN_TX_GetStates_Cyclic
FUNCTION_BLOCK FB_CAN_TX_GetStates_Cyclic
VAR_INPUT
	cycleTimeIn_mSec: UDINT:= 3000;
END_VAR
VAR_OUTPUT
END_VAR
VAR
	CAN_Tx_Faults: ifmRCAN.CAN_Tx;
	CAN_Tx_StatusState: ifmRCAN.CAN_Tx;
	CAN_Tx_BatteryVoltage: ifmRCAN.CAN_Tx;
	

	
		// Cyclic states reading
	b_BatteryStateFrameReceived: BOOL; // when received the next state (Faults) will be asked (can will be sended)
	b_FaultsFrameReceived: BOOL; // next State (Motor Controller)
	b_MotorControlFrameReceived: BOOL;
	RS_CyclicReadStates: Rs;
	TON_runtimeStatus: TON;
	TON_getStatusStates: TON;
	TON_getVoltage: TON;
	// Shifting of Bytes and converting from dV to V
	BYTE_TO_BITS_0: BYTE_TO_BITS;
	BYTE_TO_BITS_1: BYTE_TO_BITS;
	Buffer_To_String_0: ifmFileUtil.Buffer_To_String;
	batteryStateInProcent: REAL;
	TON_TimeToGetStates: TON;
	RS_StatesReadingActive: RS;
	RS_ReadingFaultsState: RS;
	RS_ReadingMotorControllerState: RS;
	RS_ReadingBatteryState: RS;
	RS_ReadingFauslts: RS;
	CAN_Tx_RunTimeStatus1: ifmRCAN.CAN_Tx;
	TON_CycleTime: TON;
	TON_runtimeStatus2: TON;
	CAN_Tx_RunTimeStatus2: ifmRCAN.CAN_Tx;
	RS_TX_StatusState: RS;
	RS_TX_BatteryVoltage: RS;
	RS_TX_RunTimeStatus1: RS;
	RS_TX_RunTimeStatus2: RS;
	TON_runtimeStatusOff: TON;
	RS_TX_Faults: RS;
	CTU_BatteryVoltageRequestDelay: CTU;
END_VAR
VAR // added by the converter: edge detectors and wires of the graphical bodies
    _rt1, _rt2, _rt3, _rt4, _rt5, _rt6, _rt7, _rt8, _rt9 : R_TRIG;
END_VAR

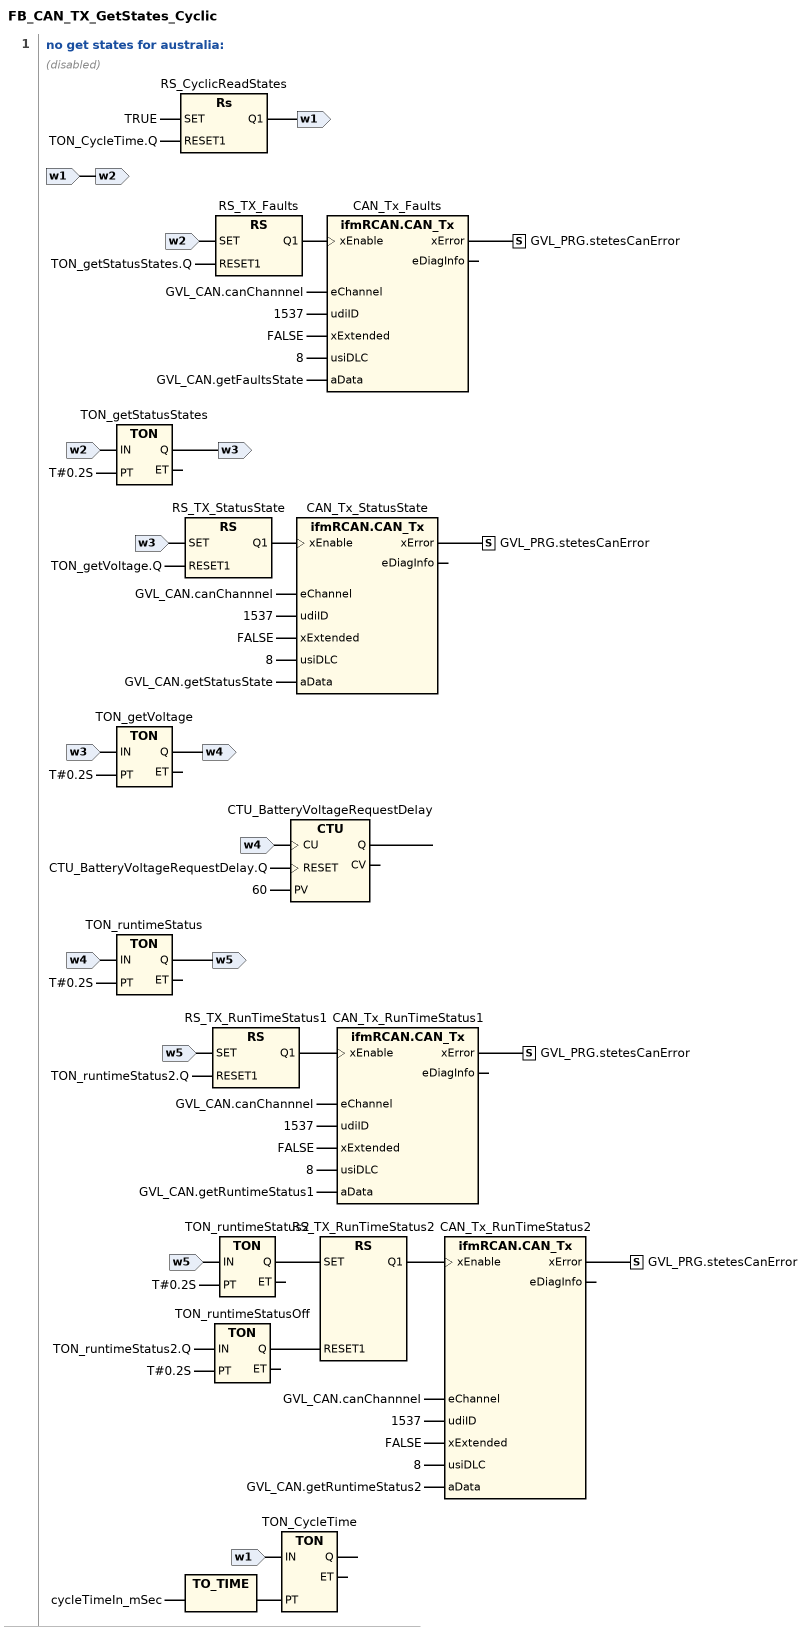
// NETWORK 1 (disabled)
// label: no get states for australia
// RS_CyclicReadStates(SET := TRUE, RESET1 := TON_CycleTime.Q); // Rs
// RS_TX_Faults(SET := RS_CyclicReadStates.Q1, RESET1 := TON_getStatusStates.Q); // RS
// _rt1(CLK := RS_TX_Faults.Q1);
// CAN_Tx_Faults(
//     xEnable := _rt1.Q,
//     eChannel := GVL_CAN.canChannnel,
//     udiID := 1537,
//     xExtended := FALSE,
//     usiDLC := 8,
//     aData := GVL_CAN.getFaultsState); // ifmRCAN.CAN_Tx
// GVL_PRG.stetesCanError S= CAN_Tx_Faults.xError;
// TON_getStatusStates(IN := RS_CyclicReadStates.Q1, PT := T#0.2S); // TON
// RS_TX_StatusState(SET := TON_getStatusStates.Q, RESET1 := TON_getVoltage.Q); // RS
// _rt2(CLK := RS_TX_StatusState.Q1);
// CAN_Tx_StatusState(
//     xEnable := _rt2.Q,
//     eChannel := GVL_CAN.canChannnel,
//     udiID := 1537,
//     xExtended := FALSE,
//     usiDLC := 8,
//     aData := GVL_CAN.getStatusState); // ifmRCAN.CAN_Tx
// GVL_PRG.stetesCanError S= CAN_Tx_StatusState.xError;
// TON_getVoltage(IN := TON_getStatusStates.Q, PT := T#0.2S); // TON
// _rt3(CLK := TON_getVoltage.Q);
// _rt4(CLK := CTU_BatteryVoltageRequestDelay.Q);
// CTU_BatteryVoltageRequestDelay(CU := _rt3.Q, RESET := _rt4.Q, PV := 60); // CTU
// TON_runtimeStatus(IN := TON_getVoltage.Q, PT := T#0.2S); // TON
// RS_TX_RunTimeStatus1(SET := TON_runtimeStatus.Q, RESET1 := TON_runtimeStatus2.Q); // RS
// _rt5(CLK := RS_TX_RunTimeStatus1.Q1);
// CAN_Tx_RunTimeStatus1(
//     xEnable := _rt5.Q,
//     eChannel := GVL_CAN.canChannnel,
//     udiID := 1537,
//     xExtended := FALSE,
//     usiDLC := 8,
//     aData := GVL_CAN.getRuntimeStatus1); // ifmRCAN.CAN_Tx
// GVL_PRG.stetesCanError S= CAN_Tx_RunTimeStatus1.xError;
// TON_runtimeStatus2(IN := TON_runtimeStatus.Q, PT := T#0.2S); // TON
// TON_runtimeStatusOff(IN := TON_runtimeStatus2.Q, PT := T#0.2S); // TON
// RS_TX_RunTimeStatus2(SET := TON_runtimeStatus2.Q, RESET1 := TON_runtimeStatusOff.Q); // RS
// _rt6(CLK := RS_TX_RunTimeStatus2.Q1);
// CAN_Tx_RunTimeStatus2(
//     xEnable := _rt6.Q,
//     eChannel := GVL_CAN.canChannnel,
//     udiID := 1537,
//     xExtended := FALSE,
//     usiDLC := 8,
//     aData := GVL_CAN.getRuntimeStatus2); // ifmRCAN.CAN_Tx
// GVL_PRG.stetesCanError S= CAN_Tx_RunTimeStatus2.xError;
// TON_CycleTime(IN := RS_CyclicReadStates.Q1, PT := TO_TIME(cycleTimeIn_mSec)); // TON

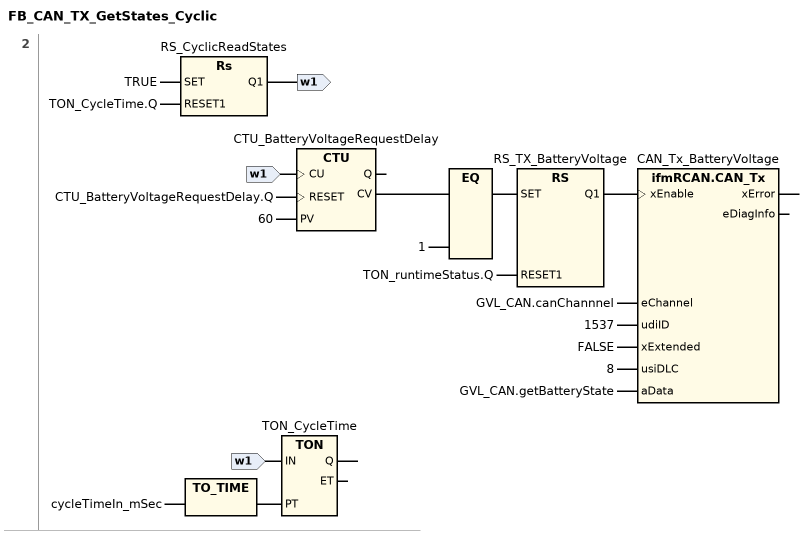
// NETWORK 2
RS_CyclicReadStates(SET := TRUE, RESET1 := TON_CycleTime.Q); // Rs
_rt7(CLK := RS_CyclicReadStates.Q1);
_rt8(CLK := CTU_BatteryVoltageRequestDelay.Q);
CTU_BatteryVoltageRequestDelay(CU := _rt7.Q, RESET := _rt8.Q, PV := 60); // CTU
RS_TX_BatteryVoltage(SET := CTU_BatteryVoltageRequestDelay.CV = 1, RESET1 := TON_runtimeStatus.Q); // RS
_rt9(CLK := RS_TX_BatteryVoltage.Q1);
CAN_Tx_BatteryVoltage(
    xEnable := _rt9.Q,
    eChannel := GVL_CAN.canChannnel,
    udiID := 1537,
    xExtended := FALSE,
    usiDLC := 8,
    aData := GVL_CAN.getBatteryState); // ifmRCAN.CAN_Tx
TON_CycleTime(IN := RS_CyclicReadStates.Q1, PT := TO_TIME(cycleTimeIn_mSec)); // TON

END_FUNCTION_BLOCK

// Device/Application/FBs/location/locatoinSimulation
FUNCTION_BLOCK locatoinSimulation
VAR_INPUT
		EN: BOOL;
		turning: BOOL;
		bMovingDirection: BOOL; // 0: forword 1: Back
		bRowDirection: BOOL;
		countOfRows: USINT;
		canRecived_CurrentRowNumber: USINT := 255;
		cr_turningInToNextRow: BOOL;
		frontClosed: BOOL;
		backClosed: BOOL;
		nextRotationAngle: BOOL:=FALSE; // 1: right 0: left
		
END_VAR
VAR_OUTPUT
	calculatedCurrentRowNumber: USINT;
	antXYa: ARRAY[0..2] OF UINT:=[0,0,0];
END_VAR
VAR
	pixelsBetween2Rows : USINT := 100;
	xAnt: INT;
	yAnt: INT;
	xAntStart: INT := 476;
	dXant: SINT := 1;
	previosRowNumber: UINT:= 0 ;
	TON_1: TON;
	RS_Turning: RS;
	TON_2: TON;
	CTU_0: CTU;
	TON_3: TON;
	TON_4: TON;
	RS_1: RS;
	RS_2: RS;
	RS_3: RS;
	CTU_CurrentRowNumber: CTU;
	calculatedNextRowsignal_FT: BOOL;
	turningBetween2Rows: BOOL;
	nextRow: BOOL;
	TOGGLE_turningBetween2Rows: TOGGLE;
	SR_closedRow: SR;
	RS_Rotate: RS;
	TON_Rotate: TON;
	dAlpha: REAL:= 1.8;
	alphaAnt: REAL:=0;
	TOGGLE_Turningdirection: TOGGLE;
END_VAR
VAR // added by the converter: edge detectors and wires of the graphical bodies
    _rt1, _rt2, _rt3, _rt4, _rt5, _rt6, _rt7, _rt8, _rt9, _rt10, _rt11, _rt12, _rt13, _rt14, _rt15, _rt16, _rt17 : R_TRIG;
    _w1, _w2 : BOOL;
    _ft1, _ft2 : F_TRIG;
END_VAR

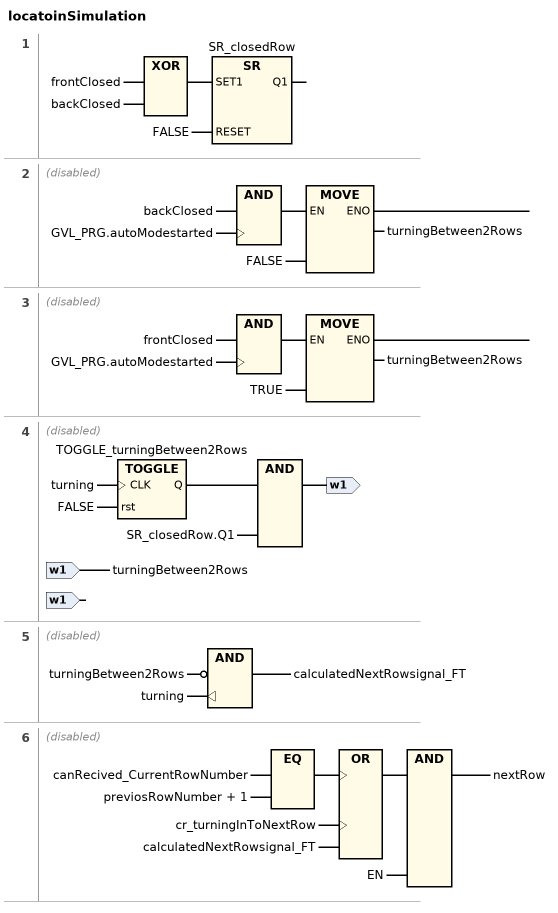
// NETWORK 1
SR_closedRow(SET1 := frontClosed XOR backClosed, RESET := FALSE); // SR

// NETWORK 2 (disabled)
// _rt1(CLK := GVL_PRG.autoModestarted);
// IF backClosed AND _rt1.Q THEN turningBetween2Rows := FALSE; END_IF

// NETWORK 3 (disabled)
// _rt2(CLK := GVL_PRG.autoModestarted);
// IF frontClosed AND _rt2.Q THEN turningBetween2Rows := TRUE; END_IF

// NETWORK 4 (disabled)
// _rt3(CLK := turning);
// TOGGLE_turningBetween2Rows(CLK := _rt3.Q, rst := FALSE); // TOGGLE
// _w1 := TOGGLE_turningBetween2Rows.Q AND SR_closedRow.Q1;
// turningBetween2Rows := _w1;

// NETWORK 5 (disabled)
// _ft1(CLK := turning);
// calculatedNextRowsignal_FT := NOT turningBetween2Rows AND _ft1.Q;

// NETWORK 6 (disabled)
// _rt4(CLK := canRecived_CurrentRowNumber = (previosRowNumber + 1));
// _rt5(CLK := cr_turningInToNextRow);
// nextRow := (_rt4.Q OR _rt5.Q OR calculatedNextRowsignal_FT) AND EN;

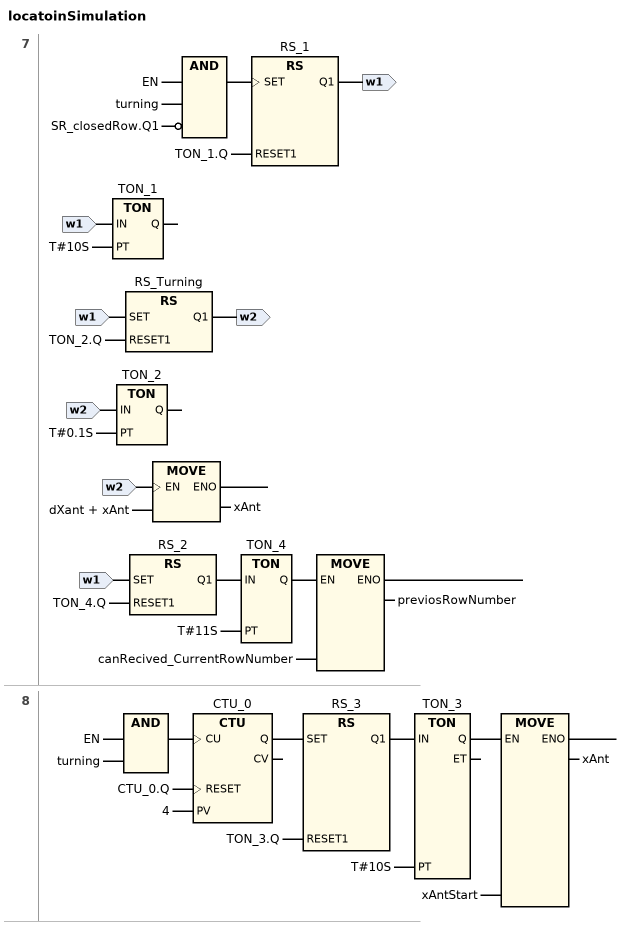
// NETWORK 7
_rt6(CLK := EN AND turning AND NOT SR_closedRow.Q1);
RS_1(SET := _rt6.Q, RESET1 := TON_1.Q); // RS
TON_1(IN := RS_1.Q1, PT := T#10S); // TON
RS_Turning(SET := RS_1.Q1, RESET1 := TON_2.Q); // RS
TON_2(IN := RS_Turning.Q1, PT := T#0.1S); // TON
_rt7(CLK := RS_Turning.Q1);
IF _rt7.Q THEN xAnt := dXant + xAnt; END_IF
RS_2(SET := RS_1.Q1, RESET1 := TON_4.Q); // RS
TON_4(IN := RS_2.Q1, PT := T#11S); // TON
IF TON_4.Q THEN previosRowNumber := canRecived_CurrentRowNumber; END_IF

// NETWORK 8
_rt8(CLK := EN AND turning);
_rt9(CLK := CTU_0.Q);
CTU_0(CU := _rt8.Q, RESET := _rt9.Q, PV := 4); // CTU
RS_3(SET := CTU_0.Q, RESET1 := TON_3.Q); // RS
TON_3(IN := RS_3.Q1, PT := T#10S); // TON
IF TON_3.Q THEN xAnt := xAntStart; END_IF

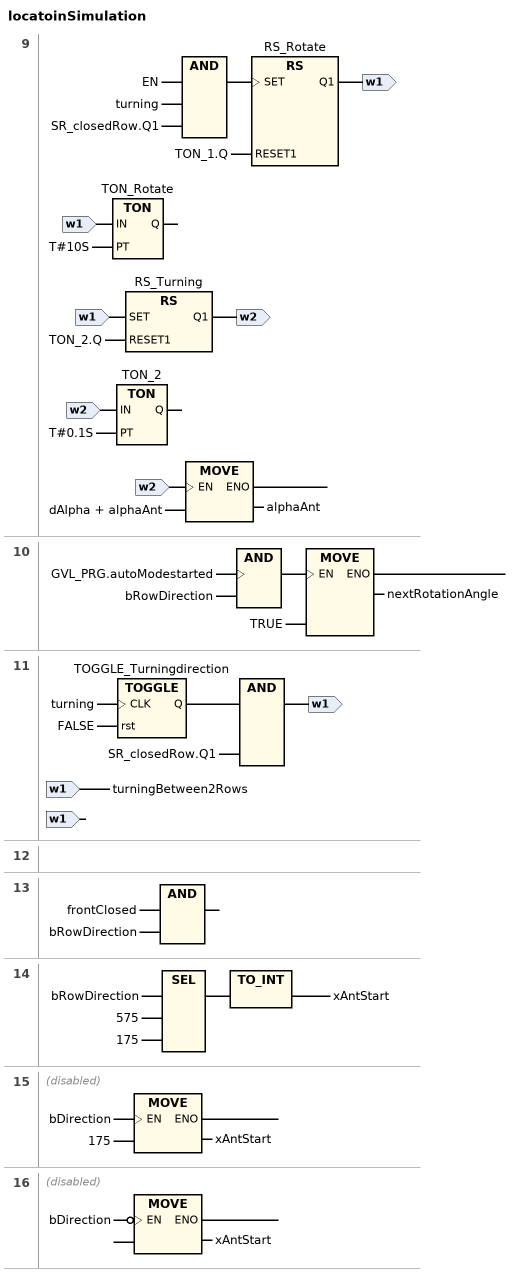
// NETWORK 9
_rt10(CLK := EN AND turning AND SR_closedRow.Q1);
RS_Rotate(SET := _rt10.Q, RESET1 := TON_1.Q); // RS
TON_Rotate(IN := RS_Rotate.Q1, PT := T#10S); // TON
RS_Turning(SET := RS_Rotate.Q1, RESET1 := TON_2.Q); // RS
TON_2(IN := RS_Turning.Q1, PT := T#0.1S); // TON
_rt11(CLK := RS_Turning.Q1);
IF _rt11.Q THEN alphaAnt := dAlpha + alphaAnt; END_IF

// NETWORK 10
_rt12(CLK := GVL_PRG.autoModestarted);
_rt13(CLK := _rt12.Q AND bRowDirection);
IF _rt13.Q THEN nextRotationAngle := TRUE; END_IF

// NETWORK 11
_rt14(CLK := turning);
TOGGLE_Turningdirection(CLK := _rt14.Q, rst := FALSE); // TOGGLE
_w2 := TOGGLE_Turningdirection.Q AND SR_closedRow.Q1;
turningBetween2Rows := _w2;

// NETWORK 12

// NETWORK 13
(* frontClosed AND bRowDirection; result not used *)

// NETWORK 14
xAntStart := TO_INT(SEL(bRowDirection, 575, 175));

// NETWORK 15 (disabled)
// _rt15(CLK := bDirection);
// IF _rt15.Q THEN xAntStart := 175; END_IF

// NETWORK 16 (disabled)
// _rt16(CLK := NOT bDirection);
// IF _rt16.Q THEN xAntStart := ???; END_IF

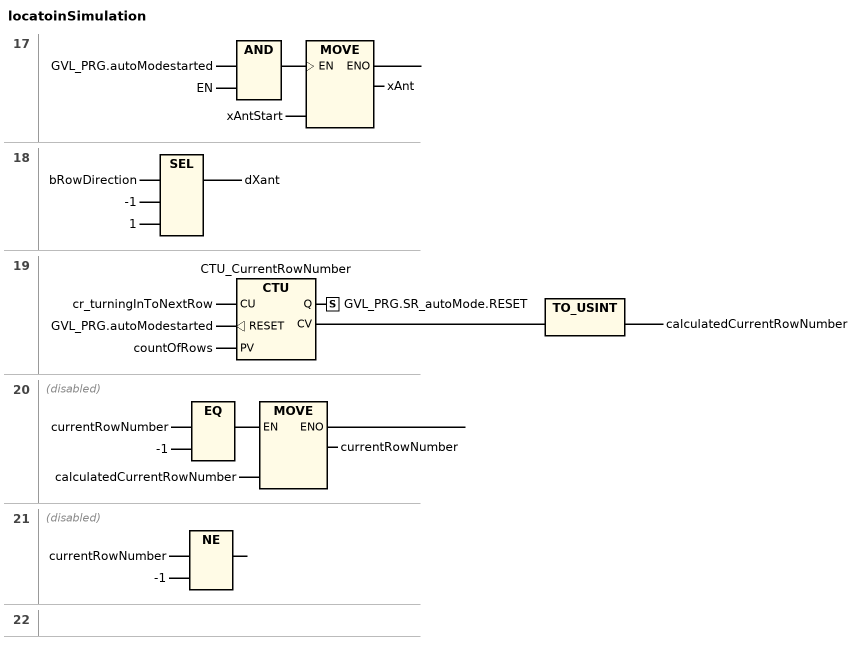
// NETWORK 17
_rt17(CLK := GVL_PRG.autoModestarted AND EN);
IF _rt17.Q THEN xAnt := xAntStart; END_IF

// NETWORK 18
dXant := SEL(bRowDirection, -1, 1);

// NETWORK 19
_ft2(CLK := GVL_PRG.autoModestarted);
CTU_CurrentRowNumber(CU := cr_turningInToNextRow, RESET := _ft2.Q, PV := countOfRows); // CTU
GVL_PRG.SR_autoMode.RESET S= CTU_CurrentRowNumber.Q;
calculatedCurrentRowNumber := TO_USINT(CTU_CurrentRowNumber.CV);

// NETWORK 20 (disabled)
// IF currentRowNumber = -1 THEN currentRowNumber := calculatedCurrentRowNumber; END_IF

// NETWORK 21 (disabled)
// (* currentRowNumber <> -1; result not used *)

// NETWORK 22

END_FUNCTION_BLOCK

// Device/Application/can/FB_CAN_RX
// Voltage >= 53.6 V:
// 8 column Estimate: 100% SoC (Full, after a short rest period after charging)
// Voltage approx. 53.2 V - 53.5 V:
// 7 column Estimate: ~90% - 99% SoC (Very full) here 90%
// Voltage approx. 52.8 V - 53.1 V:
// 6 Estimate: ~70% - 90% SoC (The 80% range could be roughly placed here)
// Voltage approx. 52.0 V - 52.7 V:
// 4 Estimate: ~30% - 70% SoC (The flattest part of the curve, very inaccurate) here 50%
// Voltage approx. 51.2 V - 51.9 V: 
// 2 Estimate: ~15% - 30% SoC (Voltage starts to drop slightly) here 20%
// Voltage approx. 50.0 V - 51.1 V:
// 1 Estimate: ~10% - 15% SoC (Voltage drops more noticeably) here 10%
// Voltage < 50.0 V:
// 0 Estimate: ~0% - 10% SoC (Near the discharge limit) here 0%

FUNCTION_BLOCK FB_CAN_RX
VAR_INPUT
END_VAR
VAR_OUTPUT
	turning: BOOL:= FALSE;
	r_batteryVoltage: REAL:=0.0;
	strMotorControllerState: STRING(100);
	strFaultsState: STRING;
END_VAR
VAR
	CAN_Rx_State: ifmRCAN.CAN_Rx;
		// Battery state
	
	batteryStateFrameMask: ARRAY [0..7] OF USINT := [00,13,33,0,0,0,0,0];
	b_BatteryStateFrameReceived : BOOL;
	// Faults
	faultsState: STRING;
	faultsFrameMask: ARRAY [0..7] OF USINT := [0,18,33,0,0,0,0,0];
	
	b_FaultsFrameReceived : BOOL;
	
	// Motor controller state
	MotorControllerStateFrameMask: ARRAY [0..7] OF USINT := [0,17,33,0,0,0,0,0];
	FB_DefineMotorControllerState_0: FB_DefineMotorControllerState;
	b_MotorControlFrameReceived : BOOL;
	b_accelerationFrameReceived_1: bool;
	
	// location
	
	startTurningFrameMask: ARRAY [0..7] OF USINT := [0,127,33,1,0,0,0,0];
	//stopTurningFrameMask: ARRAY [0..7] OF USINT := [0,127,33,2,0,0,0,0];
	voltageOffset: INT := 0;
	battery100: BOOL;
	battery90: BOOL;
	battery80: BOOL;
	battery50: BOOL;
	battery20: BOOL;
	battery10: BOOL;
	battery0: BOOL;
	
	//CAN_Rx_jetson: ifmRCAN.CAN_Rx;

	FB_SoC_FromVoltage_0: FB_SoC_FromVoltage;
END_VAR

VAR_OUTPUT RETAIN
	
END_VAR
VAR RETAIN
		ar_BatteryState: ARRAY [0..1] OF BYTE :=[0,0];
		ar_acceleration: ARRAY [0..1] OF BYTE :=[0,0];
		ar_FaultsState: ARRAY [0..1] OF USINT;
		MotorControllerState: USINT:= 0;
END_VAR
VAR // added by the converter: edge detectors and wires of the graphical bodies
    _w1, _w2, _w3, _w4, _w5, _w6, _w7, _w8, _w9, _w10, _w11, _w12, _w13, _w14, _w15 : BOOL;
    _rt1, _rt2, _rt3, _rt4, _rt5, _rt6, _rt7, _rt8, _rt9 : R_TRIG;
END_VAR

